# EPICS autosave request: iocBoot/ioclogitechF710/UserSeq.req
$(P)$(R)$(SEQ).LNK1
$(P)$(R)$(SEQ).LNK2
$(P)$(R)$(SEQ).LNK3
$(P)$(R)$(SEQ).LNK4
$(P)$(R)$(SEQ).LNK5
$(P)$(R)$(SEQ).LNK6
$(P)$(R)$(SEQ).LNK7
$(P)$(R)$(SEQ).LNK8
$(P)$(R)$(SEQ).LNK9

$(P)$(R)$(SEQ).DO1
$(P)$(R)$(SEQ).DO2
$(P)$(R)$(SEQ).DO3
$(P)$(R)$(SEQ).DO4
$(P)$(R)$(SEQ).DO5
$(P)$(R)$(SEQ).DO6
$(P)$(R)$(SEQ).DO7
$(P)$(R)$(SEQ).DO8
$(P)$(R)$(SEQ).DO9
